// Gets the current date and time (now)
FUNCTION GetDateTime : DATE_AND_TIME
VAR
	fbSystemTime : GETSYSTEMTIME;
	timeAsFileTime : T_FILETIME;
END_VAR

fbSystemTime(timeLoDW => timeAsFileTime.dwLowDateTime, timeHiDW => timeAsFileTime.dwHighDateTime);
GetDateTime := FILETIME_TO_DT(timeAsFileTime);

END_FUNCTION

(* stored: Version 1.1.0.1, ProductVersion 3.1.4024.11
   POU GetDateTime: Id {d98f9110-38cf-48a3-9cd0-78009fa76cb7}, SpecialFunc None *)
